PROGRAM MAIN
VAR
END_VAR

END_PROGRAM

(* stored: Version 1.1.0.1
   POU MAIN: Id {9e1d1d90-3633-4afb-a345-9ceb368b7520} *)
